// TIA Portal V20 export
DATA_BLOCK "PMC_FaultWord"   // DB385
// stored: InstanceOfName CITI_Logic.zPMC_FaultWord, InstanceOfType FB, Namespace CITI_Logic
"CITI_Logic.zPMC_FaultWord"
   // VAR_OUTPUT
   //    TMP_PMC_FaultIndex : Int;
   // END_VAR
   // VAR_IN_OUT
   //    FaultWords : Array[0..499] of Word;
   // END_VAR
   // VAR
   //    sFaultWords : Array[0..499] of Word;
   //    sDestArray : Array[1..8000] of Bool;
   // END_VAR
BEGIN
END_DATA_BLOCK
